{attribute 'linkalways'} 
{attribute 'no_explicit_call' := 'This FB is a CLASS and must be accessed using methods or properties'}
{attribute 'enable_dynamic_creation'}
FUNCTION_BLOCK Node_F_VN_DrawRectangle EXTENDS VisionNode
VAR
    nTopLeftX : _UDINT(0);
    nTopLeftY : _UDINT(0);
    nBottomRightX : _UDINT(0);
    nBottomRightY : _UDINT(0);
    ipDestImage : _ITcVnImage;
    aColor : _TcVnVector4_LREAL;
    nThickness : _DINT(1);
    hrPrev : _HRESULT(S_OK);
	hresult : _HRESULT(S_OK);
END_VAR

METHOD PUBLIC  Clone : I_Node
VAR
	pNode : POINTER TO Node_F_VN_DrawRectangle;
END_VAR
pNode := __NEW(Node_F_VN_DrawRectangle);
Clone := pNode^;
END_METHOD

METHOD FB_init : BOOL
VAR_INPUT
	bInitRetains : BOOL; // if TRUE, the retain variables are initialized (warm start / cold start)
	bInCopyCode : BOOL;  // if TRUE, the instance afterwards gets moved into the copy code (online change)
END_VAR
AddParameter('nTopLeftX', nTopLeftX);
AddParameter('nTopLeftY', nTopLeftY);
AddParameter('nBottomRightX', nBottomRightX);
AddParameter('nBottomRightY', nBottomRightY);
AddInput('ipDestImage', ipDestImage);
AddInput('aColor', aColor);
AddParameter('nThickness', nThickness);
AddInput('hrPrev', hrPrev);
AddOutput('ipDestImage', ipDestImage);
AddOutput('hresult',hresult);
END_METHOD

METHOD PROTECTED OnExecute
hresult.Value := F_VN_DrawRectangle(
    nTopLeftX := nTopLeftX.Value,
    nTopLeftY := nTopLeftY.Value,
    nBottomRightX := nBottomRightX.Value,
    nBottomRightY := nBottomRightY.Value,
	ipDestImage := ipDestImage.Value,
    aColor := aColor.Value,
    nThickness := nThickness.Value,
	hrPrev:= hrPrev.Value);
END_METHOD

METHOD PUBLIC PreExecutionCheck
VAR_INPUT
	Check : I_PreExecutionChecks;
END_VAR
Check.IsTrue(ipDestImage.IsValid, 'ipDestImage must contain an image');
Check.IsTrue(nThickness.Value <> 0, 'nThickness must be non-zero');
END_METHOD

END_FUNCTION_BLOCK

(* stored: Version 1.1.0.1, ProductVersion 3.1.4024.15
   POU Node_F_VN_DrawRectangle: Id {0ccc153b-cfcc-0982-1ac5-b296deadb32b}, SpecialFunc None
   Folder Constructor: Id {6fa0a212-1fa3-0b75-2731-ae3dae961510}
   Method Clone: Id {7b60ae7e-a101-0545-2b80-973ea64c22f2}
   Method FB_init: Id {b5d34f25-a7a1-0d1f-064b-1ffa1c7e281a}
   Method OnExecute: Id {1550631a-32f3-005b-1ee9-660e25c777e9}
   Method PreExecutionCheck: Id {68a964e8-51af-063b-0f0a-424e037e45ab} *)
